FUNCTION_BLOCK FB_TimeIntegrator
VAR_INPUT
	fIn 		: LREAL;
	fStepTime 	: LREAL;
	fInit 		: LREAL;
	bEnableLimits : BOOL := FALSE;
	fMinVal		: LREAL;
	fMaxVal		: LREAL;
END_VAR
VAR_OUTPUT
	fOut : LREAL := fInit;
END_VAR
VAR
END_VAR


IF bEnableLimits THEN
	fOut := LIMIT(fMinVal, fOut + fIn*fStepTime, fMaxVal);
ELSE
	fOut := fOut + fIn*fStepTime;	
END_IF

END_FUNCTION_BLOCK

(* stored: Version 1.1.0.1, ProductVersion 3.1.4024.9
   POU FB_TimeIntegrator: Id {b9c66d37-7bb0-4d0a-adb1-9688c6d8363a}, SpecialFunc None *)
